FUNCTION F_LogContext : I_ContextBuilder
VAR_STAT
	aTaskContext		: ARRAY[1..SIZEOF(TwinCAT_SystemInfoVarList._TaskInfo)/SIZEOF(PlcTaskSystemInfo)] OF FB_ContextBuilder;
END_VAR

F_LogContext := aTaskContext[Tc2_System.GETCURTASKINDEXEX()].Clear();

END_FUNCTION

(* stored: Version 1.1.0.1, ProductVersion 3.1.4024.0
   POU F_LogContext: Id {15bc0808-4d58-45ab-93cf-1a8d645eec0b}, SpecialFunc None *)
